(* PLC project SafeLOGIC-1, BrAutomation SafeDESIGNER  5.12.2.0 *)
(* stored: companyURL http://www.br-automation.com, creationDateTime Sun Apr 04 16:55:07 2021 *)

PROGRAM Main
  VAR  (* added by the conversion: wires and edge detectors of the diagram *)
    _AND_S71_OUT : SAFEBOOL;
    _OR_S134_OUT : SAFEBOOL;
  END_VAR

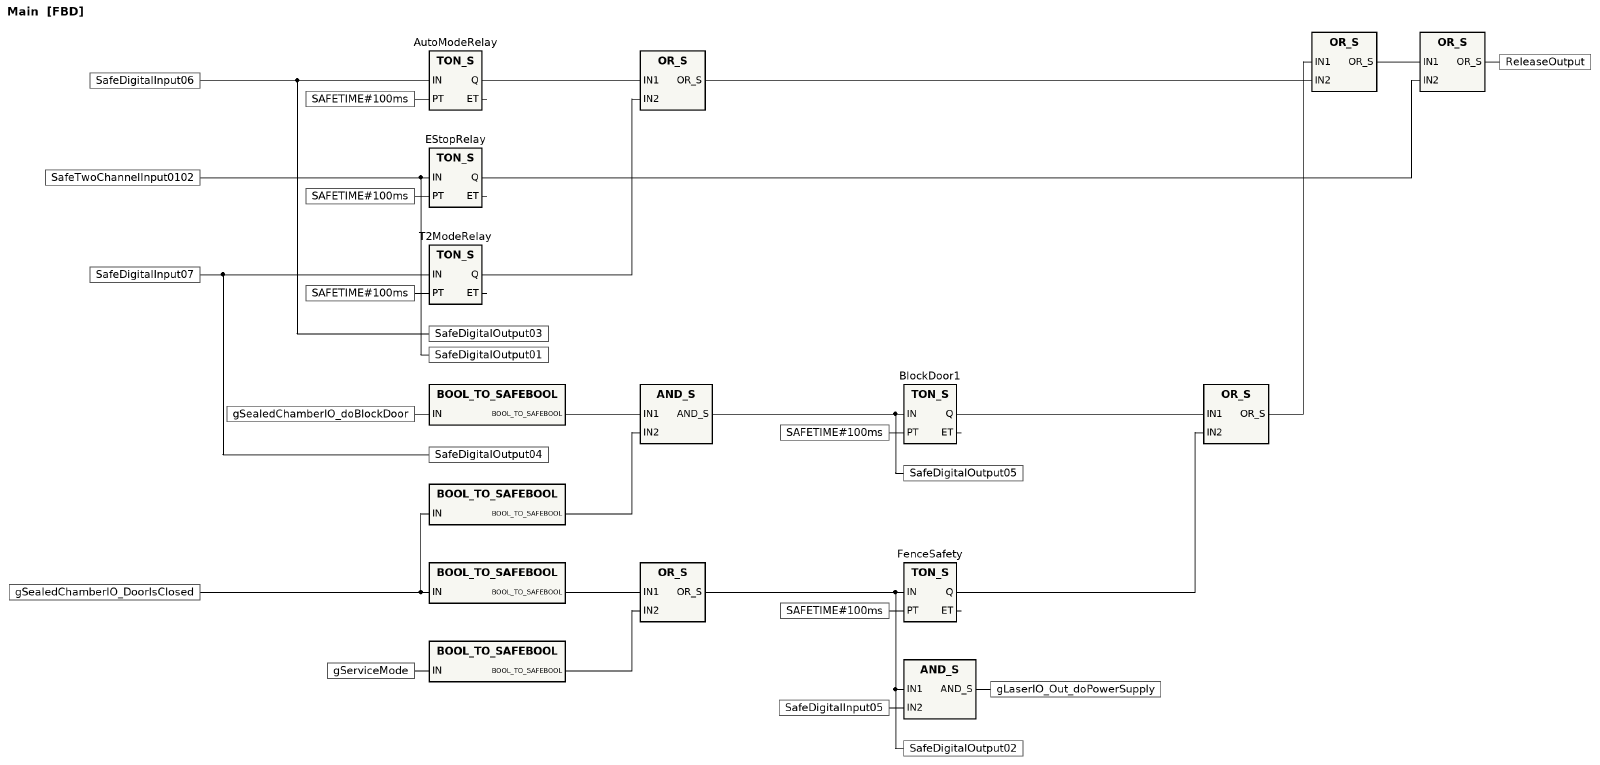
(* FBD diagram, written out as Structured Text *)
_AND_S71_OUT := AND_S(BOOL_TO_SAFEBOOL(gSealedChamberIO_doBlockDoor), BOOL_TO_SAFEBOOL(gSealedChamberIO_DoorIsClosed));
SafeDigitalOutput05 := _AND_S71_OUT;
_OR_S134_OUT := OR_S(BOOL_TO_SAFEBOOL(gSealedChamberIO_DoorIsClosed), BOOL_TO_SAFEBOOL(gServiceMode));
SafeDigitalOutput02 := _OR_S134_OUT;
gLaserIO_Out_doPowerSupply := AND_S(_OR_S134_OUT, SafeDigitalInput05);
SafeDigitalOutput03 := SafeDigitalInput06;
SafeDigitalOutput04 := SafeDigitalInput07;
BlockDoor1(IN := _AND_S71_OUT, PT := SAFETIME#100ms);
FenceSafety(IN := _OR_S134_OUT, PT := SAFETIME#100ms);
AutoModeRelay(IN := SafeDigitalInput06, PT := SAFETIME#100ms);
T2ModeRelay(IN := SafeDigitalInput07, PT := SAFETIME#100ms);
EStopRelay(IN := SafeTwoChannelInput0102, PT := SAFETIME#100ms);
ReleaseOutput := OR_S(OR_S(OR_S(BlockDoor1.Q, FenceSafety.Q), OR_S(AutoModeRelay.Q, T2ModeRelay.Q)), EStopRelay.Q);
SafeDigitalOutput01 := SafeTwoChannelInput0102;
END_PROGRAM
